// TIA Portal V20 export
// export: Created 2026-04-28T10:05:07.5794276Z, ExportSetting WithDefaults, DisplayName Totally Integrated Automation Portal, DisplayVersion V20, DisplayName TIA Portal Openness, DisplayVersion V20, DisplayName TIA Portal Version Control Interface, DisplayVersion V20, DisplayName SINAMICS Startdrive Advanced, DisplayVersion V20, DisplayName SINAMICS Startdrive G130, G150, S120, S150, SINAMICS MV, G220, S200, S210, DisplayVersion V20, DisplayName SINAMICS Startdrive G110M, G120, G120C, G120D, G120P, G115D, DisplayVersion V20, DisplayName STEP 7 Professional, DisplayVersion V20, DisplayName STEP 7 Safety, DisplayVersion V20, DisplayName WinCC Basic/Comfort/Advanced, DisplayVersion V20, DisplayName WinCC Unified, DisplayVersion V20
TYPE "KonfigurationProzess"
// stored: IsFailsafeCompliant false
   STRUCT
      i30_RangZeile1 : Int;
      i30_RangZeile2 : Int;
      i30_RangZeile3 : Int;
      i30_RangZeile4 : Int;
      i30_RangZeile5 : Int;
      i10_RangZeile1 : Int;
      i10_RangZeile2 : Int;
      i10_RangZeile3 : Int;
      i10_RangZeile4 : Int;
      i10_RangZeile5 : Int;
      i10_RangZeile6 : Int;
      i60_RangZeile1 : Int;
      i60_RangZeile2 : Int;
      i60_RangZeile3 : Int;
      i60_RangZeile4 : Int;
      i60_RangZeile5 : Int;
      i60_RangZeile6 : Int;
      i60_RangZeile7 : Int;
      i60_RangZeile8 : Int;
      i60_RangZeile9 : Int;
      i60_RangZeile10 : Int;
      i60_RangZeile11 : Int;
      i60_RangZeile12 : Int;
      i20_RangZeile1 : Int;
      i20_RangZeile2 : Int;
      i20_RangZeile3 : Int;
      i20_RangZeile4 : Int;
      i20_RangZeile5 : Int;
      i20_RangZeile6 : Int;
      i20_RangZeile7 : Int;
      i40_RangZeile1 : Int;
      i40_RangZeile2 : Int;
      i40_RangZeile3 : Int;
      i40_RangZeile4 : Int;
      i50_RangZeile1 : Int;
      i50_RangZeile2 : Int;
      i50_RangZeile3 : Int;
      i50_RangZeile4 : Int;
      i50_RangZeile5 : Int;
      i50_RangZeile6 : Int;
      i50_RangZeile7 : Int;
      i50_RangZeile8 : Int;
      i50_RangZeile9 : Int;
      i50_RangZeile10 : Int;
      i50_RangZeile11 : Int;
      i50_RangZeile12 : Int;
   END_STRUCT;
END_TYPE
